{attribute 'linkalways'} 
{attribute 'no_explicit_call' := 'This FB is a CLASS and must be accessed using methods or properties'}
{attribute 'enable_dynamic_creation'}
FUNCTION_BLOCK Node_ContainerType_Vector_ULINT EXTENDS Node
VAR
    out : _GUID;
END_VAR

METHOD PUBLIC  Clone : I_Node
VAR
	pNode : POINTER TO Node_ContainerType_Vector_ULINT;
END_VAR
pNode := __NEW(Node_ContainerType_Vector_ULINT);
Clone := pNode^;
END_METHOD

METHOD FB_init : BOOL
VAR_INPUT
	bInitRetains : BOOL; // if TRUE, the retain variables are initialized (warm start / cold start)
	bInCopyCode : BOOL;  // if TRUE, the instance afterwards gets moved into the copy code (online change)
END_VAR
AddOutput('out', out);
END_METHOD

METHOD PROTECTED OnExecute
out.Value := ContainerType_Vector_ULINT;
END_METHOD

END_FUNCTION_BLOCK

(* stored: Version 1.1.0.1, ProductVersion 3.1.4026.17
   POU Node_ContainerType_Vector_ULINT: Id {b2011aeb-007a-0078-2f4f-9c78d81fd969}, SpecialFunc None
   Folder Constructor: Id {2a2f14e7-4d5b-0b85-1c8c-da7e7cf02a21}
   Method Clone: Id {39f3c727-5529-02b5-3c77-d86a069f8a18}
   Method FB_init: Id {eb5d1e8e-a8f5-038c-0d59-7a7e18f4244c}
   Method OnExecute: Id {3c3d3eb3-c392-0ef3-293b-1f9275950d8b} *)
